ABB RobotStudio station: UiS_E458_nov18.rspag

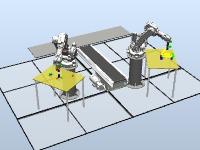
--- station ---
Station UiS_E458_nov18 (saved by RobotStudio 6.6.7701.1025)
Controller Rudolf, task T_ROB1: task frame (RAPID world) sits at (10, 680, 720) mm, rotated rx 0 ry 0 rz -30 deg in the station
Controller Norbert, task T_ROB1: task frame (RAPID world) sits at (-305, -752, 720) mm, rotated rx 0 ry 0 rz 30 deg in the station
Controller Norbert
  mechanical unit ROB_1: Norbert, 6 joints, base frame (0, 0, 0) mm
Controller Rudolf
  mechanical unit ROB_1: Rudolf, 6 joints, base frame (0, 0, 0) mm
Layout (positions relative to the parent item):
  - PedestalR [part, from Libraries\Pedestal.rslib] at (10, 680, 0) mm, rotated rx 0 ry 0 rz 150 deg
  - PedestalN [part, from Libraries\Pedestal.rslib] at (-305, -752, 0) mm, rotated rx 0 ry 0 rz -150 deg
  - Conveyor [part, from Libraries\Conveyor.rslib] at (-998.97, -64.27, 615.81) mm, rotated rx 90 ry 0 rz -90 deg
  - Windowtable [part]
  - TableN [part, from Libraries\Desk.rslib] at (-421.89, -1050.54, 0) mm, rotated rx 0 ry 0 rz -60 deg
  - TableR [part, from Libraries\Desk.rslib] at (193.4, 1497.66, 0) mm, rotated rx 0 ry 0 rz -120 deg
  - SC_Gripper [smart component, from Libraries\SC_Gripper.rslib] at (74.9, -1110.01, 1042.25) mm, rotated rx 180 ry 0 rz 120 deg
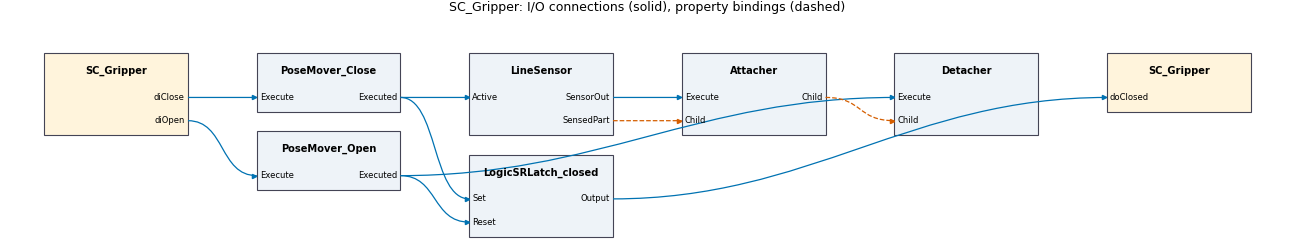
      connections:
        SC_Gripper.diClose -> PoseMover_Close.Execute
        PoseMover_Close.Executed -> LogicSRLatch_closed.Set
        SC_Gripper.diOpen -> PoseMover_Open.Execute
        PoseMover_Open.Executed -> LogicSRLatch_closed.Reset
        LogicSRLatch_closed.Output -> SC_Gripper.doClosed
        PoseMover_Close.Executed -> LineSensor.Active
        LineSensor.SensorOut -> Attacher.Execute
        PoseMover_Open.Executed -> Detacher.Execute
        LineSensor.SensedPart => Attacher.Child
        Attacher.Child => Detacher.Child
    - tGripper [mechanism, from Libraries\SC_Gripper.rslib] at (0, 0, 0) mm; joint values [0.006, 0.006] (rad or m)
    - PoseMover_Close [smart component, from Components\PoseMover.rslib]
        properties: Mechanism=tGripper; Pose=2; Duration=1
    - LogicSRLatch_closed [smart component, from Components\LogicSRLatch.rslib]
    - PoseMover_Open [smart component, from Components\PoseMover.rslib]
        properties: Mechanism=tGripper; Pose=1; Duration=1
    - LineSensor [smart component, from Components\LineSensor.rslib]
        properties: Start=[-5.20417042793042E-18 -0.0255 0.10825]; End=[-2.47198095326695E-17 0.0255 0.10825]; Radius=0.002; SensedPart=Puck1; SensedPoint=[0.126558441162109 -0.849249755859375 0.744]
      - _sensorPart_ [part]
    - Attacher [smart component, from Components\Attacher.rslib]
        properties: Parent=tGripper; Flange=0; Child=Puck1; Mount=false; Offset=[0 0 0]; Orientation=[0 0 0]
    - Detacher [smart component, from Components\Detacher.rslib]
        properties: Child=Puck1; KeepPosition=true
  - UISpenholder [mechanism, from Libraries\UISpenholder.rslib] at (483.21, 1099.62, 1138) mm, rotated rx 180 ry 0 rz 150 deg
  - Norbert [mechanism, from Robots\IRB140_6_81_C_G_03.rslib] at (-305, -752, 720) mm, rotated rx 0 ry 0 rz 30 deg; joint values [-1.2793, 0.5463, 0.2528, 0, 0.7717, 0.2915] (rad or m)
  - Rudolf [mechanism, from Robots\IRB140_6_81_C_G_03.rslib] at (10, 680, 720) mm, rotated rx 0 ry 0 rz -30 deg; joint values [1.249, 0.6446, -0.2193, 0, 1.1455, 1.249] (rad or m)
  - Puck1 [part] at (-98.25, -1210.1, 728) mm, rotated rx 0 ry 0 rz -60 deg
Attachment: TableN is attached to PedestalN
Attachment: TableR is attached to PedestalR
Attachment: SC_Gripper is attached to Norbert / Link6
Attachment: UISpenholder is attached to Rudolf / Link6
Station signals: DI doClose, DI doOpen
Station logic (signal -> signal, property => property):
  Norbert.doOpen -> SC_Gripper.diOpen
  Norbert.doClose -> SC_Gripper.diClose
  SC_Gripper.doClosed -> Norbert.diClosed

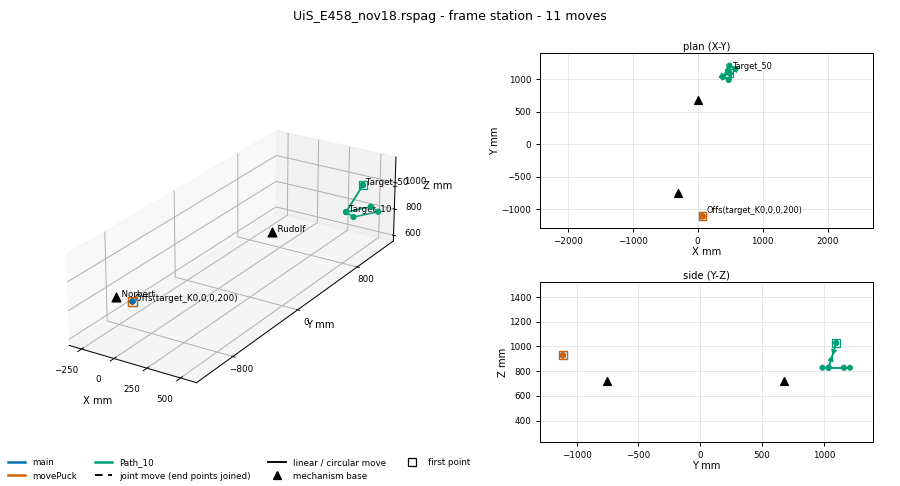
[picture p0: tool path of UiS_E458_nov18.rspag in frame station, 11 of 21 moves have a stored position in this frame; points joined in program order, loops and branches not executed]
--- Backups/Norbert/RAPID/TASK1/PROGMOD/E458GripperTest.mod ---
MODULE E458GripperTest
    ! Module for testing gripper, UiS KS Nov. 29, 2018

    ! wobj in the middle of the table, x-axis along short side of table, y-axis along long axis
	TASK PERS wobjdata wobjTableN:=[FALSE,TRUE,"",[[150,-500,8],[0.707106781,0,0,-0.707106781]],[[0,0,0],[1,0,0,0]]];

    ! robtargets
	CONST robtarget target_K0:=[[0,0,0],[0,1,0,0],[0,0,0,0],[9E9,9E9,9E9,9E9,9E9,9E9]];
	CONST robtarget target_K1:=[[0,-200,0],[0,1,0,0],[0,0,0,0],[9E9,9E9,9E9,9E9,9E9,9E9]];
	CONST robtarget target_K2:=[[-200,200,0],[0,1,0,0],[0,0,0,0],[9E9,9E9,9E9,9E9,9E9,9E9]];

	PROC main()
	    MoveL Offs(target_K0, 0, 0, 200),v500,z10,tGripper\WObj:=wobjTableN;
	    movePuck;
	ENDPROC

    PROC movePuck()
	    MoveJ Offs(target_K0, 0, 0, 200),v500,z10,tGripper\WObj:=wobjTableN;
        WaitTime 1.0;
        getPuck(target_K1);
        putPuck(target_K2);
	    MoveJ Offs(target_K0, 0, 0, 200),v500,z10,tGripper\WObj:=wobjTableN;
        WaitTime 1.0;
        getPuck(target_K2);
        putPuck(target_K1);
	    MoveJ Offs(target_K0, 0, 0, 200),v500,z10,tGripper\WObj:=wobjTableN;
        WaitTime 1.0;
    ENDPROC

    PROC getPuck(robtarget pos)
        MoveJ Offs(pos, 0, 0, 200),v500,z50,tGripper\WObj:=wobjTableN;
        MoveJ Offs(pos, 0, 0, 50),v200,z10,tGripper\WObj:=wobjTableN;
	    MoveL Offs(pos, 0, 0, 10),v50,fine,tGripper\WObj:=wobjTableN;
        closeGripper(TRUE);
	    MoveL Offs(pos, 0, 0, 50),v50,z10,tGripper\WObj:=wobjTableN;
        MoveJ Offs(pos, 0, 0, 200),v200,z50,tGripper\WObj:=wobjTableN;
    ENDPROC

    PROC putPuck(robtarget pos)
        MoveJ Offs(pos, 0, 0, 200),v500,z50,tGripper\WObj:=wobjTableN;
        MoveJ Offs(pos, 0, 0, 50),v200,z10,tGripper\WObj:=wobjTableN;
	    MoveL Offs(pos, 0, 0, 10),v50,fine,tGripper\WObj:=wobjTableN;
        closeGripper(FALSE);
	    MoveL Offs(pos, 0, 0, 50),v50,z10,tGripper\WObj:=wobjTableN;
        MoveJ Offs(pos, 0, 0, 200),v200,z50,tGripper\WObj:=wobjTableN;
    ENDPROC

ENDMODULE

--- Backups/Norbert/RAPID/TASK1/PROGMOD/gripper.mod ---
MODULE gripper
    ! Module for gripper, UiS KS Nov. 29, 2018

    PERS tooldata tGripper:=[TRUE,[[0,0,114.25],[0,0,0,1]],[1,[-0.095984607,0.082520613,38.69176324],[1,0,0,0],0,0,0]];

    ! for virtual controller Norbert (simulation)
    PROC closeGripper(bool state)
        WaitTime 0.2;
        IF state=TRUE THEN
          SetDO doClose, 1;
          SetDO doOpen, 0;
        ELSEIF state=FALSE THEN
          SetDO doClose, 0;
          SetDO doOpen, 1;
        ENDIF
        WaitTime 1.2;
    ENDPROC

   ! for actual or physical robot Norbert
   ! Note that different IO signals are used here
!    PROC closeGripper(bool state)
!        WaitTime 0.1;
!        IF state=TRUE THEN
!          setDO doGripOpen, 0;
!          setDO doGripClose, 1;
!        ELSEIF state=FALSE THEN
!          setDO doGripOpen, 1;
!          setDO doGripClose, 0;
!        ENDIF
!        WaitTime 0.2;
!    ENDPROC

ENDMODULE

--- Backups/Norbert/RAPID/TASK1/SYSMOD/LINKEDM.sys ---
%%%
  VERSION:1
  LANGUAGE:ENGLISH
%%%

MODULE LINKEDM (SYSMODULE)

! FOLLOWER
!     Name of electronically linked follower axis used by operator at teach pendent.
      PERS string l_f_axis_name{5}       :=  ["",  "", "", "", ""];

!     Name of the mechanical unit for follower axis.
      PERS string l_f_mecunt_n{5}  :=  ["", "", "", "", ""];

!     Linked follower axis number in the mechanical unit (first axis in mech. unit is number 1).
      PERS num l_f_axis_no{5}      :=  [0,          0,   0,  0,  0];

! MASTER
!     Name of the mechanical unit for linked master axis.
      PERS string l_m_mecunt_n{5} :=  ["", "", "", "", ""];

!     Linked master axis number in the mechanical unit (first axis in mech. unit is number 1).
!     See axis number table in documentation for different master mechanical units.
      PERS num l_m_axis_no{5}     :=  [0,  0,  0,  0,  0];

! POSITION OFFSET
!     The increase of the allowed offset position between the master and follower
!     positions, used when starting AUTO mode. As soon as the offset is decreased
!     the old configurated parameter is used.
!     Example: 3 => the configurated value of allowed offset is increased 3 times.
      PERS num offset_ratio{5}       :=  [10,  10,   10,  10,  10];

! SPEED RATIO
!     Speed_ratio used in AUTO and JOG modes [ very_slow   slow    normal    fast]
!     Value 1 = max allowed manual speed.
      CONST num speed_ratio {20}      := [0.01, 0.01, 0.01, 0.01, 0.01,
                                          0.05, 0.05, 0.05, 0.05, 0.05,
                                          0.20, 0.20, 0.20, 0.20, 0.20,
                                          1.00, 1.00, 1.00, 1.00, 1.00];

! STEP SIZE
!     Displacement position used in JOG mode for each activation of positive or
!     negative movement.                  [very_short    short   normal   long]
!     Unit degees or meter.
      CONST num displacement {20}     := [0.001, 0.001, 0.001, 0.001, 0.001,
                                          0.005, 0.005, 0.005, 0.005, 0.005,
                                          0.020, 0.020, 0.020, 0.020, 0.020,
                                          0.100, 0.100, 0.100, 0.100, 0.100];


!-------------------------------------------------------------
 PROC Linked_m ()
      Linked_m_exe ;
 ENDPROC
ENDMODULE

--- Backups/Rudolf/RAPID/TASK1/PROGMOD/E458PenTest.mod ---
MODULE E458PenTest
    ! Module for testing pen, UiS KS Nov. 29, 2018

    ! wobj in the middle of the table
    TASK PERS wobjdata wobjTableR:=[FALSE,TRUE,"",[[150,500,8],[1,0,0,0]],[[0,0,0],[1,0,0,0]]];
    PERS tooldata tSimplePen:=[TRUE,[[0,0,110],[1,0,0,0]],[1,[0,0,1],[1,0,0,0],0,0,0]];

    CONST robtarget Target_10:=[[0,0,100],[0,0,1,0],[0,0,0,0],[9E9,9E9,9E9,9E9,9E9,9E9]];
    CONST robtarget Target_20:=[[100,0,100],[0,0,1,0],[0,0,0,0],[9E9,9E9,9E9,9E9,9E9,9E9]];
    CONST robtarget Target_30:=[[100,200,100],[0,0,1,0],[0,0,0,0],[9E9,9E9,9E9,9E9,9E9,9E9]];
    CONST robtarget Target_40:=[[0,200,100],[0,0,1,0],[0,0,0,0],[9E9,9E9,9E9,9E9,9E9,9E9]];
    CONST robtarget Target_50:=[[50,100,300],[0,0,1,0],[0,0,0,0],[9E9,9E9,9E9,9E9,9E9,9E9]];

    PROC main()
        Path_10;
    ENDPROC

    PROC Path_10()
        MoveL Target_50,v500,z10,tSimplePen\WObj:=wobjTableR;
        MoveL Target_10,v500,z10,tSimplePen\WObj:=wobjTableR;
        MoveL Target_20,v500,z10,tSimplePen\WObj:=wobjTableR;
        MoveL Target_30,v500,z10,tSimplePen\WObj:=wobjTableR;
        MoveL Target_40,v500,z10,tSimplePen\WObj:=wobjTableR;
        MoveL Target_10,v500,z10,tSimplePen\WObj:=wobjTableR;
        MoveL Target_50,v500,z10,tSimplePen\WObj:=wobjTableR;
    ENDPROC

ENDMODULE

--- Backups/Norbert/SYSPAR/EIO.cfg ---
EIO:CFG_1.0:6:1::
#
EIO_SIGNAL:

      -Name "diClosed" -SignalType "DI" -Access "All"

      -Name "doClose" -SignalType "DO" -Access "All"

      -Name "doOpen" -SignalType "DO" -Access "All"
